{attribute 'GeneratedUsingTerminal: KL6224-0001'}
{attribute addProperty BoxType "KL6224-0001"}
{attribute addProperty Id "StatusAT %I*UINT0Parameter_InAT %I*UDINT0State_Ch1AT %I*USINT0State_Ch2AT %I*USINT0State_Ch3AT %I*USINT0State_Ch4AT %I*USINT0Data_In_0AT %I*USINT0Data_In_1AT %I*USINT0Data_In_2AT %I*USINT0Data_In_3AT %I*USINT0Data_In_4AT %I*USINT0Data_In_5AT %I*USINT0Data_In_6AT %I*USINT0Data_In_7AT %I*USINT0Data_In_8AT %I*USINT0Data_In_9AT %I*USINT0Data_In_10AT %I*USINT0Data_In_11AT %I*USINT0Data_In_12AT %I*USINT0Data_In_13AT %I*USINT0ControlAT %Q*UINT0Parameter_OutAT %Q*UDINT0Data_Out_0AT %Q*USINT0Data_Out_1AT %Q*USINT0Data_Out_2AT %Q*USINT0Data_Out_3AT %Q*USINT0Data_Out_4AT %Q*USINT0Data_Out_5AT %Q*USINT0Data_Out_6AT %Q*USINT0Data_Out_7AT %Q*USINT0Data_Out_8AT %Q*USINT0Data_Out_9AT %Q*USINT0Data_Out_10AT %Q*USINT0Data_Out_11AT %Q*USINT0Data_Out_12AT %Q*USINT0Data_Out_13AT %Q*USINT0Data_Out_14AT %Q*USINT0Data_Out_15AT %Q*USINT0Data_Out_16AT %Q*USINT0Data_Out_17AT %Q*USINT0"}
{attribute addProperty CRC "139671556"}
{attribute addProperty Size "0"}
TYPE Channel_08533804 :
STRUCT
	{attribute addProperty Name "Status"}
	Status AT %I* : UINT;
	{attribute addProperty Name "Parameter_In"}
	Parameter_In AT %I* : UDINT;
	{attribute addProperty Name "State_Ch1"}
	State_Ch1 AT %I* : USINT;
	{attribute addProperty Name "State_Ch2"}
	State_Ch2 AT %I* : USINT;
	{attribute addProperty Name "State_Ch3"}
	State_Ch3 AT %I* : USINT;
	{attribute addProperty Name "State_Ch4"}
	State_Ch4 AT %I* : USINT;
	{attribute addProperty Name "Data_In_0"}
	Data_In_0 AT %I* : USINT;
	{attribute addProperty Name "Data_In_1"}
	Data_In_1 AT %I* : USINT;
	{attribute addProperty Name "Data_In_2"}
	Data_In_2 AT %I* : USINT;
	{attribute addProperty Name "Data_In_3"}
	Data_In_3 AT %I* : USINT;
	{attribute addProperty Name "Data_In_4"}
	Data_In_4 AT %I* : USINT;
	{attribute addProperty Name "Data_In_5"}
	Data_In_5 AT %I* : USINT;
	{attribute addProperty Name "Data_In_6"}
	Data_In_6 AT %I* : USINT;
	{attribute addProperty Name "Data_In_7"}
	Data_In_7 AT %I* : USINT;
	{attribute addProperty Name "Data_In_8"}
	Data_In_8 AT %I* : USINT;
	{attribute addProperty Name "Data_In_9"}
	Data_In_9 AT %I* : USINT;
	{attribute addProperty Name "Data_In_10"}
	Data_In_10 AT %I* : USINT;
	{attribute addProperty Name "Data_In_11"}
	Data_In_11 AT %I* : USINT;
	{attribute addProperty Name "Data_In_12"}
	Data_In_12 AT %I* : USINT;
	{attribute addProperty Name "Data_In_13"}
	Data_In_13 AT %I* : USINT;
	{attribute addProperty Name "Control"}
	Control AT %Q* : UINT;
	{attribute addProperty Name "Parameter_Out"}
	Parameter_Out AT %Q* : UDINT;
	{attribute addProperty Name "Data_Out_0"}
	Data_Out_0 AT %Q* : USINT;
	{attribute addProperty Name "Data_Out_1"}
	Data_Out_1 AT %Q* : USINT;
	{attribute addProperty Name "Data_Out_2"}
	Data_Out_2 AT %Q* : USINT;
	{attribute addProperty Name "Data_Out_3"}
	Data_Out_3 AT %Q* : USINT;
	{attribute addProperty Name "Data_Out_4"}
	Data_Out_4 AT %Q* : USINT;
	{attribute addProperty Name "Data_Out_5"}
	Data_Out_5 AT %Q* : USINT;
	{attribute addProperty Name "Data_Out_6"}
	Data_Out_6 AT %Q* : USINT;
	{attribute addProperty Name "Data_Out_7"}
	Data_Out_7 AT %Q* : USINT;
	{attribute addProperty Name "Data_Out_8"}
	Data_Out_8 AT %Q* : USINT;
	{attribute addProperty Name "Data_Out_9"}
	Data_Out_9 AT %Q* : USINT;
	{attribute addProperty Name "Data_Out_10"}
	Data_Out_10 AT %Q* : USINT;
	{attribute addProperty Name "Data_Out_11"}
	Data_Out_11 AT %Q* : USINT;
	{attribute addProperty Name "Data_Out_12"}
	Data_Out_12 AT %Q* : USINT;
	{attribute addProperty Name "Data_Out_13"}
	Data_Out_13 AT %Q* : USINT;
	{attribute addProperty Name "Data_Out_14"}
	Data_Out_14 AT %Q* : USINT;
	{attribute addProperty Name "Data_Out_15"}
	Data_Out_15 AT %Q* : USINT;
	{attribute addProperty Name "Data_Out_16"}
	Data_Out_16 AT %Q* : USINT;
	{attribute addProperty Name "Data_Out_17"}
	Data_Out_17 AT %Q* : USINT;
END_STRUCT
END_TYPE

(* stored: Version 1.2.0.0, ProductVersion 3.1.4024.9
   DUT Channel_08533804: Id {af141f3b-08be-4b80-ab77-e6edae40613e} *)
